(* Logix 5000 project; controller Hose_HP_Test_Rig_V1 vendor 1 type 14 code 149 rev 32.11; software revision 32.00; part 4 of 10 *)
(* tags used below, declared in another part *)
   BOTTOM_NOT_CLAMPED_STN3 : BOOL;
   DOOR_CLOSE_STS_STN2 : DINT;
   DOOR_CLOSE_STS_STN3 : DINT;
   DOOR_CLOSE_STS_STN4 : DINT;
   EXHS_OK_DEL_STN2 : TIMER;
   EXHS_OK_DELSTN4 : TIMER;
   EXHS_VAL_HP_ON_STN2 : BOOL;
   EXHS_VAL_OFF_CE_STN2 : BOOL;
   EXHS_VAL_OFF_CE_STN3 : BOOL;
   EXHS_VAL_OFF_TE_STN2 : BOOL;
   EXHS_VAL_OFF_TE_STN3 : BOOL;
   ONS28 : BOOL;
   ONS29 : BOOL;
   ONS30 : BOOL;
   ONS31 : BOOL;
   ONS32 : BOOL;
   ONS33 : BOOL;
   TOP_NOT_CLAMPED_STN2 : BOOL;
   TOP_NOT_CLAMPED_STN3 : BOOL;
   TOP_NOT_CLAMPED_STN4 : BOOL;
   ABORT_STN2 : BOOL;
   ABORT_STN3 : BOOL;
   ABORT_STN4 : BOOL;
   ACT_DROP_STN2 : REAL;
   ACT_DROP_STN3 : REAL;
   ACT_DROP_STN4 : REAL;
   ACT_PR_STN2 : REAL;
   ACT_PR_STN3 : REAL;
   ACT_PR_STN4 : REAL;
   AUTO_TEST_ON_STN2 : BOOL;
   AUTO_TEST_ON_STN3 : BOOL;
   AUTO_TEST_ON_STN4 : BOOL;
   BOTTOM_CLAMP_AUTO_STN2 : BOOL;
   BOTTOM_CLAMP_AUTO_STN3 : BOOL;
   BOTTOM_CLAMP_AUTO_STN4 : BOOL;
   BOTTOM_CLAMP_BLK_STN2 : DA_SOL_FWD_SEQ;
   BOTTOM_CLAMP_BLK_STN3 : DA_SOL_FWD_SEQ;
   BOTTOM_CLAMP_BLK_STN4 : DA_SOL_FWD_SEQ;
   BOTTOM_CLAMP_OK_STN1 : BOOL;
   BOTTOM_CLAMP_OK_STN3 : BOOL;
   BOTTOM_CLAMP_OK_STN4 : BOOL;
   BOTTOM_CLAMP_PS_STN2 : ALIAS FOR Local:2:I.Data.2;
   BOTTOM_CLAMP_PS_STN3 : ALIAS FOR Local:2:I.Data.7;
   BOTTOM_CLAMP_PS_STN4 : ALIAS FOR Local:2:I.Data.12;
   BOTTOM_CLAMP_SEQ_STN2 : DINT;
   BOTTOM_CLAMP_SEQ_STN3 : DINT;
   BOTTOM_CLAMP_SEQ_STN4 : DINT;
   BOTTOM_DECLAMP_AUTO_STN2 : BOOL;
   BOTTOM_DECLAMP_AUTO_STN3 : BOOL;
   BOTTOM_DECLAMP_AUTO_STN4 : BOOL;
   BOTTOM_DECLAMP_SEQ_STN2 : DINT;
   BOTTOM_DECLAMP_SEQ_STN3 : DINT;
   BOTTOM_DECLAMP_SEQ_STN4 : DINT;
   BOTTOM_DECLMP_BLK_STN2 : DA_SOL_RET_SEQ;
   BOTTOM_DECLMP_BLK_STN3 : DA_SOL_RET_SEQ;
   BOTTOM_DECLMP_BLK_STN4 : DA_SOL_RET_SEQ;
   BOTTOM_NOT_CLAMPED_STN2 : BOOL;
   BOTTOM_NOT_CLAMPED_STN4 : BOOL;
   BOTTOM_NOT_DECLAMPED_STN2 : BOOL;
   BOTTOM_NOT_DECLAMPED_STN3 : BOOL;
   BOTTOM_NOT_DECLAMPED_STN4 : BOOL;
   CHECK_TRACE_STS_STN2 : BOOL;
   CHECK_TRACE_STS_STN3 : BOOL;
   CHECK_TRACE_STS_STN4 : BOOL;
   CLR_FAIL_ONS_STN2 : BOOL;
   CLR_FAIL_ONS_STN3 : BOOL;
   CLR_FAIL_ONS_STN4 : BOOL;
   CLR_ONS_STN2 : BOOL;
   CLR_ONS_STN3 : BOOL;
   CLR_ONS_STN4 : BOOL;
   COMP_FAULT_STN2 : BOOL;
   COMP_FAULT_STN3 : BOOL;
   COMP_FAULT_STN4 : BOOL;
   CONS_CALB_ON_STN2 : BOOL;
   CONS_CALB_ON_STN3 : BOOL;
   CONS_CALB_ON_STN4 : BOOL;
   CONS_STS_STN2 : DINT;
   CONS_STS_STN4 : DINT;
   CONS_TEST_ON : BOOL;
   CONSTRICTION_TEST_ON_STN2 : BOOL;
   CONSTRICTION_TEST_ON_STN3 : BOOL;
   CONSTRICTION_TEST_ON_STN4 : BOOL;
   DICH_STN1 : INT;
   DOOR_CLOSE_ABORT_STN2 : BOOL;
   DOOR_CLOSE_ABORT_STN3 : BOOL;
   DOOR_CLOSE_ABORT_STN4 : BOOL;
   DOOR_CLOSE_AUTO_STN2 : BOOL;
   DOOR_CLOSE_AUTO_STN3 : BOOL;
   DOOR_CLOSE_AUTO_STN4 : BOOL;
   DOOR_CLOSE_BLK_STN2 : DOOR_CLOSE;
   DOOR_CLOSE_BLK_STN3 : DOOR_CLOSE;
   DOOR_CLOSE_BLK_STN4 : DOOR_CLOSE;
   DOOR_CLOSE_OK_STN2 : BOOL;
   DOOR_CLOSE_OK_STN3 : BOOL;
   DOOR_CLOSE_OK_STN4 : BOOL;
   DOOR_CLOSE_RS_STN2 : ALIAS FOR Local:2:I.Data.0;
   DOOR_CLOSE_RS_STN3 : ALIAS FOR Local:2:I.Data.5;
   DOOR_CLOSE_RS_STN4 : ALIAS FOR Local:2:I.Data.9;
   DOOR_CLOSE_SEQ_STN2 : DA_SOL_FWD_SEQ;
   DOOR_CLOSE_SEQ_STN3 : DA_SOL_FWD_SEQ;
   DOOR_CLOSE_SEQ_STN4 : DA_SOL_FWD_SEQ;
   DOOR_NOT_CLOSED_STN2 : BOOL;
   DOOR_NOT_CLOSED_STN3 : BOOL;
   DOOR_NOT_CLOSED_STN4 : BOOL;
   DOOR_OPEN_RS_STN2 : ALIAS FOR Local:1:I.Data.15;
   DOOR_OPEN_RS_STN3 : ALIAS FOR Local:2:I.Data.4;
   DOOR_OPEN_RS_STN4 : ALIAS FOR Local:2:I.Data.10;
   DROP_CHK_SEQ_STN2 : DROP_CHECK;
   DROP_CHK_SEQ_STN3 : DROP_CHECK;
   DROP_CHK_SEQ_STN4 : DROP_CHECK;
   DROP_NOK_STN2 : BOOL;
   DROP_NOK_STN3 : BOOL;
   DROP_NOK_STN4 : BOOL;
   DROP_OK_STN2 : BOOL;
   DROP_OK_STN3 : BOOL;
   DROP_OK_STN4 : BOOL;
   DUPLICATE_STN2 : BOOL;
   DUPLICATE_STN3 : BOOL;
   DUPLICATE_STN4 : BOOL;
   EC_STN1 : DINT;
   EC_STN2 : DINT;
   EC_STN3 : DINT;
   EC_STN4 : DINT;
   EXHAUST_SET_LIM : REAL;
   EXHS_OFF_BLK_STN2 : FILL_VAL_OFF;
   EXHS_OFF_BLK_STN3 : FILL_VAL_OFF;
   EXHS_OFF_BLK_STN4 : FILL_VAL_OFF;
   EXHS_OK_DEL_STN3 : TIMER;
   EXHS_VAL_HP_ON_STN3 : BOOL;
   EXHS_VAL_HP_ON_STN4 : BOOL;
   EXHS_VAL_OFF_CE_STN4 : BOOL;
   EXHS_VAL_OFF_STN2 : BOOL;
   EXHS_VAL_OFF_STN3 : BOOL;
   EXHS_VAL_OFF_STN4 : BOOL;
   EXHS_VAL_OFF_TE_STN4 : BOOL;
   FAULTED_STN2 : BOOL;
   FAULTED_STN3 : BOOL;
   FAULTED_STN4 : BOOL;
   FILL_ACT_TIME_STN2 : REAL;
   FILL_ACT_TIME_STN3 : REAL;
   FILL_ACT_TIME_STN4 : REAL;
   FILL_CHK_STN2 : PR_CHECK;
   FILL_CHK_STN3 : PR_CHECK;
   FILL_CHK_STN4 : PR_CHECK;
   FILL_HIGH_STN2 : BOOL;
   FILL_HIGH_STN3 : BOOL;
   FILL_HIGH_STN4 : BOOL;
   FILL_HL_STN1 : REAL;
   FILL_LL_STN1 : REAL;
   FILL_LOW_STN2 : BOOL;
   FILL_LOW_STN3 : BOOL;
   FILL_LOW_STN4 : BOOL;
   FILL_SEQ_START_STN2 : SEQ_START_AND_FILL;
   FILL_SEQ_START_STN3 : SEQ_START_AND_FILL;
   FILL_SEQ_START_STN4 : SEQ_START_AND_FILL;
   FILL_SET_TIME : REAL;
   FILL_VAL_OFF_SEQ_STN2 : FILL_VAL_OFF;
   FILL_VAL_OFF_SEQ_STN3 : FILL_VAL_OFF;
   FILL_VAL_OFF_SEQ_STN4 : FILL_VAL_OFF;
   FLT_CLR_ONS_STN2 : BOOL;
   FLT_CLR_ONS_STN3 : BOOL;
   FLT_CLR_ONS_STN4 : BOOL;
   HP_P2_STN2 : REAL;
   HP_P2_STN3 : REAL;
   HP_P2_STN4 : REAL;
   HP_STS_STN2 : DINT;
   HP_STS_STN3 : DINT;
   HP_STS_STN4 : DINT;
   HP_TEST_ON : BOOL;
   INCORRECT_STN2 : BOOL;
   INCORRECT_STN3 : BOOL;
   INCORRECT_STN4 : BOOL;
   INIT_STN2 : BOOL;
   INIT_STN3 : BOOL;
   INIT_STN4 : BOOL;
   LT_COMPLETED_STN2 : BOOL;
   LT_COMPLETED_STN3 : BOOL;
   LT_COMPLETED_STN4 : BOOL;
   LT_P1_STN2 : REAL;
   LT_P1_STN3 : REAL;
   LT_P1_STN4 : REAL;
   LT_POKEYOKE_STN2 : DINT;
   LT_POKEYOKE_STN3 : DINT;
   LT_POKEYOKE_STN4 : DINT;
   MSG_STN2 : DINT;
   MSG_STN3 : DINT;
   MSG_STN4 : DINT;
   P2_STN2 : REAL;
   P2_STN3 : REAL;
   P2_STN4 : REAL;
   POKEYOKE_NOT_DONE : BOOL;
   PYOKE_LT_STN2 : BOOL;
   PYOKE_LT_STN3 : BOOL;
   PYOKE_LT_STN4 : BOOL;
   RETEST : BOOL;
   RST_EXHS_VAL_OFF_STN2 : BOOL;
   RST_EXHS_VAL_OFF_STN3 : BOOL;
   RST_EXHS_VAL_OFF_STN4 : BOOL;
   RST_SEQ_ON_STN2 : BOOL;
   RST_SEQ_ON_STN3 : BOOL;
   RST_SEQ_ON_STN4 : BOOL;
   SCAN_OK_STN2 : BOOL;
   SCAN_OK_STN3 : BOOL;
   SCAN_OK_STN4 : BOOL;
   SCR_STS : DINT[6];
   SEQ_NO_STN2 : DINT;
   SEQ_NO_STN3 : DINT;
   SEQ_NO_STN4 : DINT;
   SET_DROP : REAL;
   STAB_ACT_TIME_STN2 : REAL;
   STAB_ACT_TIME_STN3 : REAL;
   STAB_ACT_TIME_STN4 : REAL;
   STAB_CHK_STN2 : PR_CHECK;
   STAB_CHK_STN3 : PR_CHECK;
   STAB_CHK_STN4 : PR_CHECK;
   STAB_HIGH_STN2 : BOOL;
   STAB_HIGH_STN3 : BOOL;
   STAB_HIGH_STN4 : BOOL;
   STAB_LOW_STN2 : BOOL;
   STAB_LOW_STN3 : BOOL;
   STAB_LOW_STN4 : BOOL;
   STAB_SET_TIME : REAL;
   STN2_ON : BOOL;
   STN3_ON : BOOL;
   STN4_ON : BOOL;
   TEST_ACT_TIME_STN2 : REAL;
   TEST_ACT_TIME_STN3 : REAL;
   TEST_ACT_TIME_STN4 : REAL;
   TEST_SET_TIME : REAL;
   TEST_STS_STN2 : DINT;
   TEST_STS_STN3 : DINT;
   TEST_STS_STN4 : DINT;
   TEST_STS_UPDATE_STN2 : TEST_TAIL_END;
   TEST_STS_UPDATE_STN3 : TEST_TAIL_END;
   TEST_STS_UPDATE_STN4 : TEST_TAIL_END;
   TEST_VAL_OFF_STN2 : BOOL;
   TEST_VAL_OFF_STN3 : BOOL;
   TEST_VAL_OFF_STN4 : BOOL;
   TEST_VAL_ON_STN2 : BOOL;
   TEST_VAL_ON_STN3 : BOOL;
   TEST_VAL_ON_STN4 : BOOL;
   TOP_CLAMP_AUTO_STN2 : BOOL;
   TOP_CLAMP_AUTO_STN3 : BOOL;
   TOP_CLAMP_AUTO_STN4 : BOOL;
   TOP_CLAMP_BLK_STN2 : DA_SOL_FWD_SEQ;
   TOP_CLAMP_BLK_STN3 : DA_SOL_FWD_SEQ;
   TOP_CLAMP_BLK_STN4 : DA_SOL_FWD_SEQ;
   TOP_CLAMP_OK_STN2 : BOOL;
   TOP_CLAMP_OK_STN3 : BOOL;
   TOP_CLAMP_OK_STN4 : BOOL;
(* MainProgram, continued *)

ROUTINE Auto_Test_Stn2   (* ladder *)
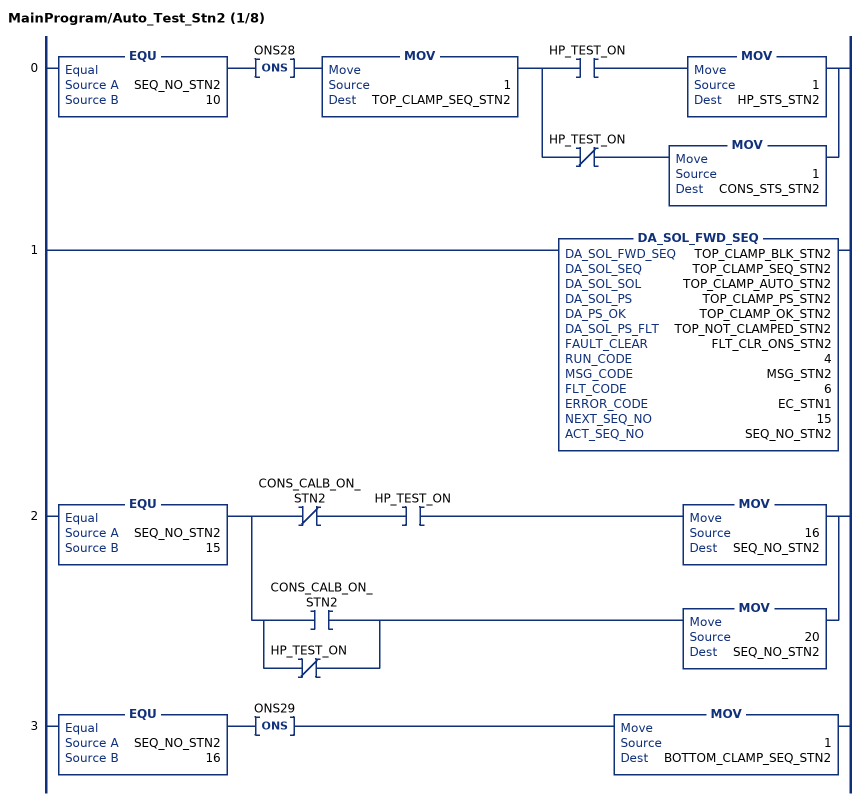
   0: EQU(SEQ_NO_STN2,10)ONS(ONS28)MOV(1,TOP_CLAMP_SEQ_STN2)[XIC(HP_TEST_ON) MOV(1,HP_STS_STN2) ,XIO(HP_TEST_ON) MOV(1,CONS_STS_STN2) ];
   1: DA_SOL_FWD_SEQ(TOP_CLAMP_BLK_STN2,TOP_CLAMP_SEQ_STN2,TOP_CLAMP_AUTO_STN2,TOP_CLAMP_PS_STN2,TOP_CLAMP_OK_STN2,TOP_NOT_CLAMPED_STN2,FLT_CLR_ONS_STN2,4,MSG_STN2,6,EC_STN1,15,SEQ_NO_STN2);
   2: EQU(SEQ_NO_STN2,15)[XIO(CONS_CALB_ON_STN2) XIC(HP_TEST_ON) MOV(16,SEQ_NO_STN2) ,[XIC(CONS_CALB_ON_STN2) ,XIO(HP_TEST_ON) ] MOV(20,SEQ_NO_STN2) ];
   3: EQU(SEQ_NO_STN2,16)ONS(ONS29)MOV(1,BOTTOM_CLAMP_SEQ_STN2);
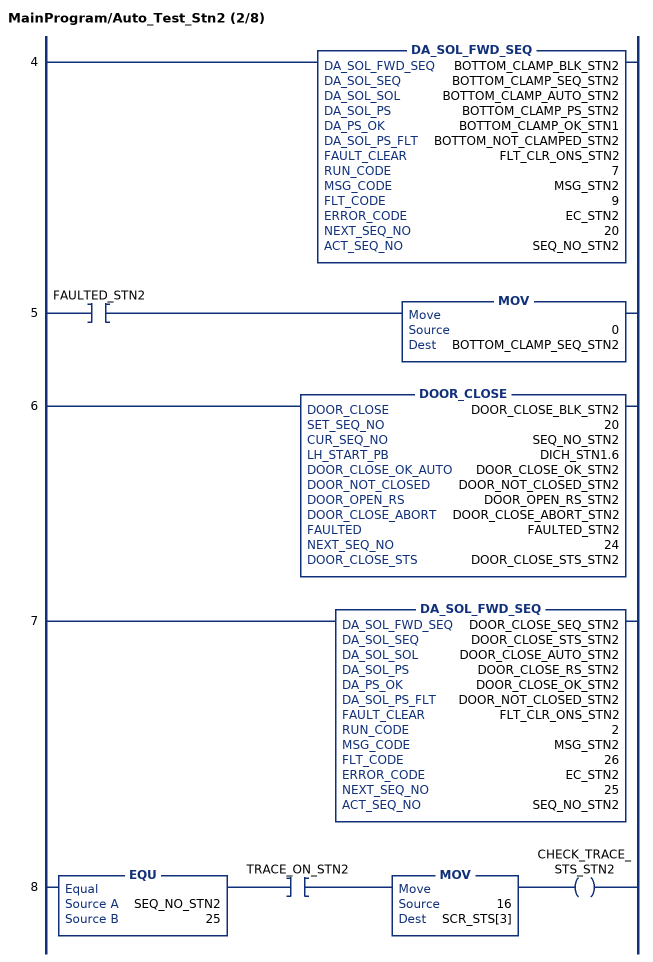
   4: DA_SOL_FWD_SEQ(BOTTOM_CLAMP_BLK_STN2,BOTTOM_CLAMP_SEQ_STN2,BOTTOM_CLAMP_AUTO_STN2,BOTTOM_CLAMP_PS_STN2,BOTTOM_CLAMP_OK_STN1,BOTTOM_NOT_CLAMPED_STN2,FLT_CLR_ONS_STN2,7,MSG_STN2,9,EC_STN2,20,SEQ_NO_STN2);
   5: XIC(FAULTED_STN2)MOV(0,BOTTOM_CLAMP_SEQ_STN2);
   6: DOOR_CLOSE(DOOR_CLOSE_BLK_STN2,20,SEQ_NO_STN2,DICH_STN1.6,DOOR_CLOSE_OK_STN2,DOOR_NOT_CLOSED_STN2,DOOR_OPEN_RS_STN2,DOOR_CLOSE_ABORT_STN2,FAULTED_STN2,24,DOOR_CLOSE_STS_STN2);
   7: DA_SOL_FWD_SEQ(DOOR_CLOSE_SEQ_STN2,DOOR_CLOSE_STS_STN2,DOOR_CLOSE_AUTO_STN2,DOOR_CLOSE_RS_STN2,DOOR_CLOSE_OK_STN2,DOOR_NOT_CLOSED_STN2,FLT_CLR_ONS_STN2,2,MSG_STN2,26,EC_STN2,25,SEQ_NO_STN2);
   8: EQU(SEQ_NO_STN2,25)XIC(TRACE_ON_STN2)MOV(16,SCR_STS[3])OTE(CHECK_TRACE_STS_STN2);
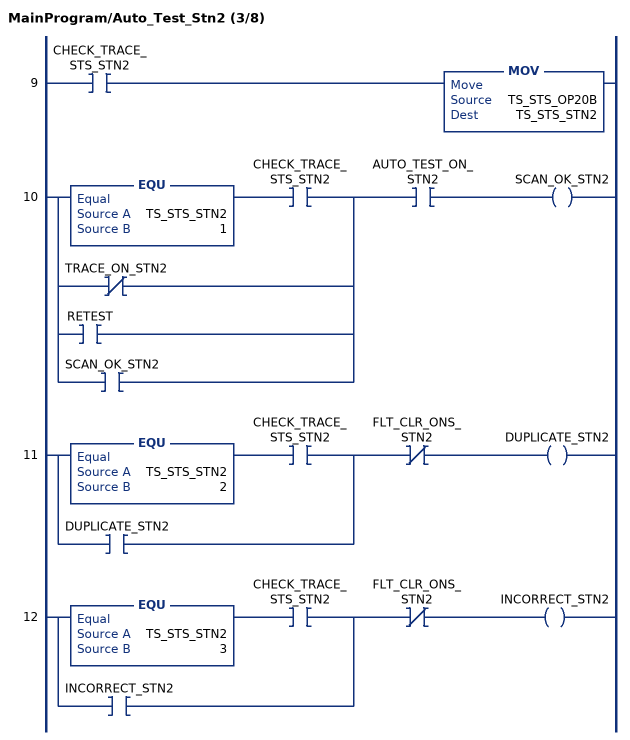
   9: XIC(CHECK_TRACE_STS_STN2)MOV(TS_STS_OP20B,TS_STS_STN2);
   10: [[EQU(TS_STS_STN2,1) XIC(CHECK_TRACE_STS_STN2) ,XIO(TRACE_ON_STN2) ,XIC(RETEST) ] ,XIC(SCAN_OK_STN2) ]XIC(AUTO_TEST_ON_STN2)OTE(SCAN_OK_STN2);
   11: [EQU(TS_STS_STN2,2) XIC(CHECK_TRACE_STS_STN2) ,XIC(DUPLICATE_STN2) ]XIO(FLT_CLR_ONS_STN2)OTE(DUPLICATE_STN2);
   12: [EQU(TS_STS_STN2,3) XIC(CHECK_TRACE_STS_STN2) ,XIC(INCORRECT_STN2) ]XIO(FLT_CLR_ONS_STN2)OTE(INCORRECT_STN2);
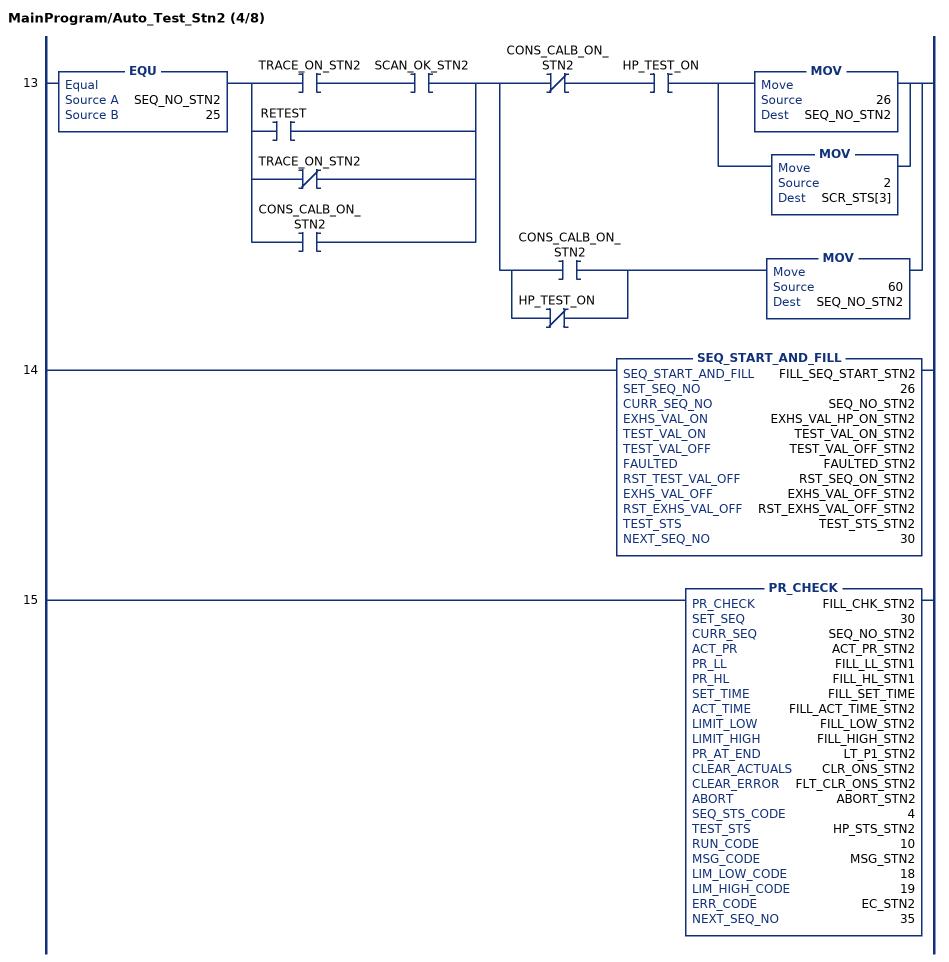
   13: EQU(SEQ_NO_STN2,25)[XIC(TRACE_ON_STN2) XIC(SCAN_OK_STN2) ,XIC(RETEST) ,XIO(TRACE_ON_STN2) ,XIC(CONS_CALB_ON_STN2) ][XIO(CONS_CALB_ON_STN2) XIC(HP_TEST_ON) [MOV(26,SEQ_NO_STN2) ,MOV(2,SCR_STS[3]) ] ,[XIC(CONS_CALB_ON_STN2) ,XIO(HP_TEST_ON) ] MOV(60,SEQ_NO_STN2) ];
   14: SEQ_START_AND_FILL(FILL_SEQ_START_STN2,26,SEQ_NO_STN2,EXHS_VAL_HP_ON_STN2,TEST_VAL_ON_STN2,TEST_VAL_OFF_STN2,FAULTED_STN2,RST_SEQ_ON_STN2,EXHS_VAL_OFF_STN2,RST_EXHS_VAL_OFF_STN2,TEST_STS_STN2,30);
   15: PR_CHECK(FILL_CHK_STN2,30,SEQ_NO_STN2,ACT_PR_STN2,FILL_LL_STN1,FILL_HL_STN1,FILL_SET_TIME,FILL_ACT_TIME_STN2,FILL_LOW_STN2,FILL_HIGH_STN2,LT_P1_STN2,CLR_ONS_STN2,FLT_CLR_ONS_STN2,ABORT_STN2,4,HP_STS_STN2,10,MSG_STN2,18,19,EC_STN2,35);
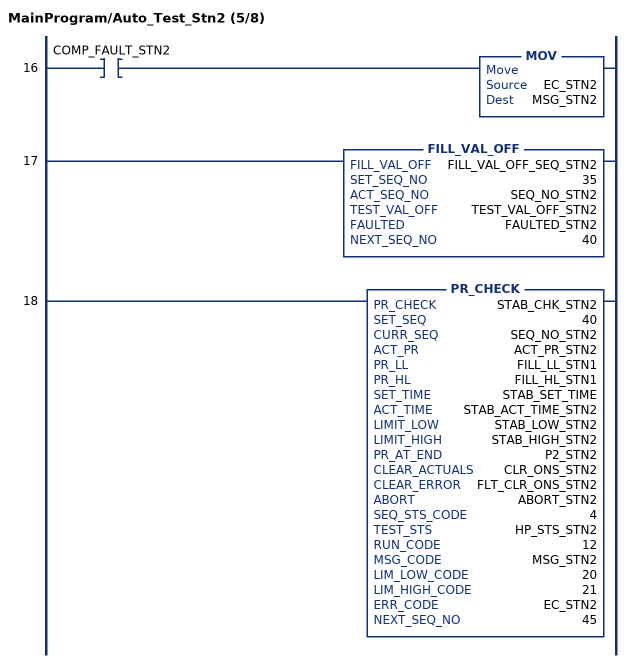
   16: XIC(COMP_FAULT_STN2)MOV(EC_STN2,MSG_STN2);
   17: FILL_VAL_OFF(FILL_VAL_OFF_SEQ_STN2,35,SEQ_NO_STN2,TEST_VAL_OFF_STN2,FAULTED_STN2,40);
   18: PR_CHECK(STAB_CHK_STN2,40,SEQ_NO_STN2,ACT_PR_STN2,FILL_LL_STN1,FILL_HL_STN1,STAB_SET_TIME,STAB_ACT_TIME_STN2,STAB_LOW_STN2,STAB_HIGH_STN2,P2_STN2,CLR_ONS_STN2,FLT_CLR_ONS_STN2,ABORT_STN2,4,HP_STS_STN2,12,MSG_STN2,20,21,EC_STN2,45);
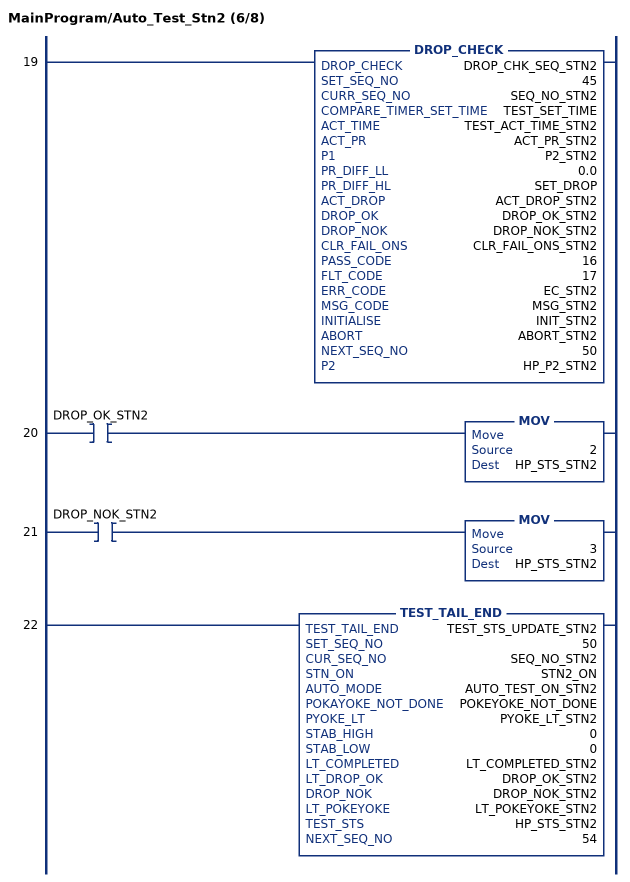
   19: DROP_CHECK(DROP_CHK_SEQ_STN2,45,SEQ_NO_STN2,TEST_SET_TIME,TEST_ACT_TIME_STN2,ACT_PR_STN2,P2_STN2,0.0,SET_DROP,ACT_DROP_STN2,DROP_OK_STN2,DROP_NOK_STN2,CLR_FAIL_ONS_STN2,16,17,EC_STN2,MSG_STN2,INIT_STN2,ABORT_STN2,50,HP_P2_STN2);
   20: XIC(DROP_OK_STN2)MOV(2,HP_STS_STN2);
   21: XIC(DROP_NOK_STN2)MOV(3,HP_STS_STN2);
   22: TEST_TAIL_END(TEST_STS_UPDATE_STN2,50,SEQ_NO_STN2,STN2_ON,AUTO_TEST_ON_STN2,POKEYOKE_NOT_DONE,PYOKE_LT_STN2,0,0,LT_COMPLETED_STN2,DROP_OK_STN2,DROP_NOK_STN2,LT_POKEYOKE_STN2,HP_STS_STN2,54);
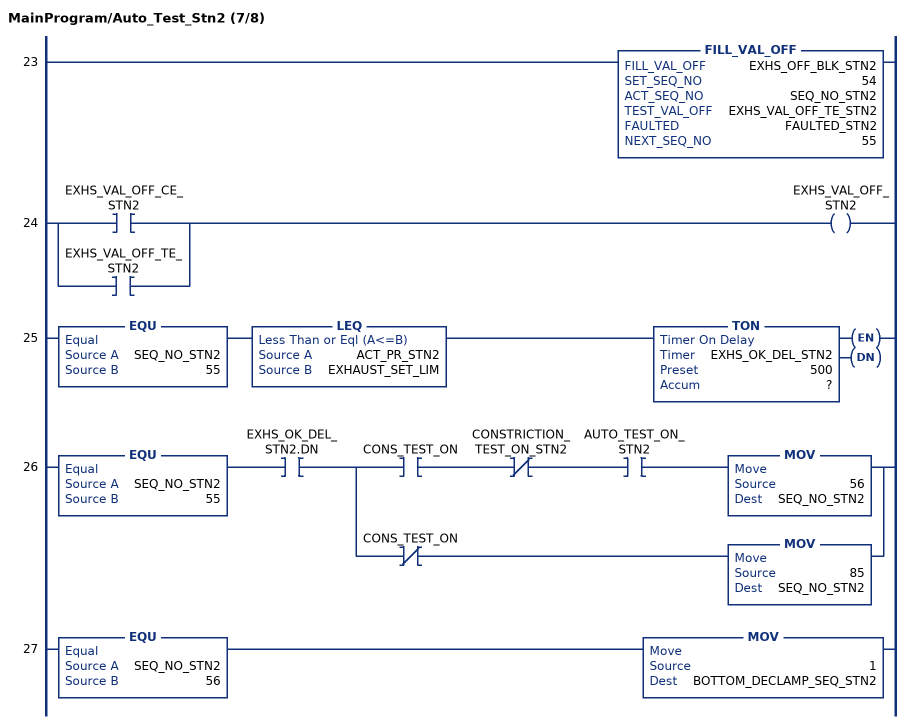
   23: FILL_VAL_OFF(EXHS_OFF_BLK_STN2,54,SEQ_NO_STN2,EXHS_VAL_OFF_TE_STN2,FAULTED_STN2,55);
   24: [XIC(EXHS_VAL_OFF_CE_STN2) ,XIC(EXHS_VAL_OFF_TE_STN2) ]OTE(EXHS_VAL_OFF_STN2);
   25: EQU(SEQ_NO_STN2,55)LEQ(ACT_PR_STN2,EXHAUST_SET_LIM)TON(EXHS_OK_DEL_STN2,?,?);
   26: EQU(SEQ_NO_STN2,55)XIC(EXHS_OK_DEL_STN2.DN)[XIC(CONS_TEST_ON) XIO(CONSTRICTION_TEST_ON_STN2) XIC(AUTO_TEST_ON_STN2) MOV(56,SEQ_NO_STN2) ,XIO(CONS_TEST_ON) MOV(85,SEQ_NO_STN2) ];
   27: EQU(SEQ_NO_STN2,56)MOV(1,BOTTOM_DECLAMP_SEQ_STN2);
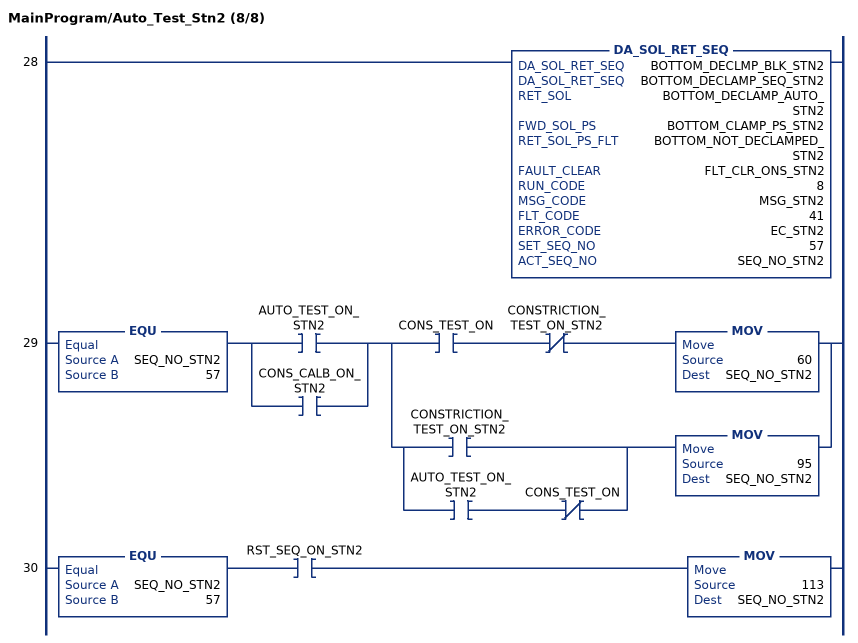
   28: DA_SOL_RET_SEQ(BOTTOM_DECLMP_BLK_STN2,BOTTOM_DECLAMP_SEQ_STN2,BOTTOM_DECLAMP_AUTO_STN2,BOTTOM_CLAMP_PS_STN2,BOTTOM_NOT_DECLAMPED_STN2,FLT_CLR_ONS_STN2,8,MSG_STN2,41,EC_STN2,57,SEQ_NO_STN2);
   29: EQU(SEQ_NO_STN2,57)[XIC(AUTO_TEST_ON_STN2) ,XIC(CONS_CALB_ON_STN2) ][XIC(CONS_TEST_ON) XIO(CONSTRICTION_TEST_ON_STN2) MOV(60,SEQ_NO_STN2) ,[XIC(CONSTRICTION_TEST_ON_STN2) ,XIC(AUTO_TEST_ON_STN2) XIO(CONS_TEST_ON) ] MOV(95,SEQ_NO_STN2) ];
   30: EQU(SEQ_NO_STN2,57)XIC(RST_SEQ_ON_STN2)MOV(113,SEQ_NO_STN2);
END_ROUTINE

ROUTINE Auto_Test_Stn3   (* ladder *)
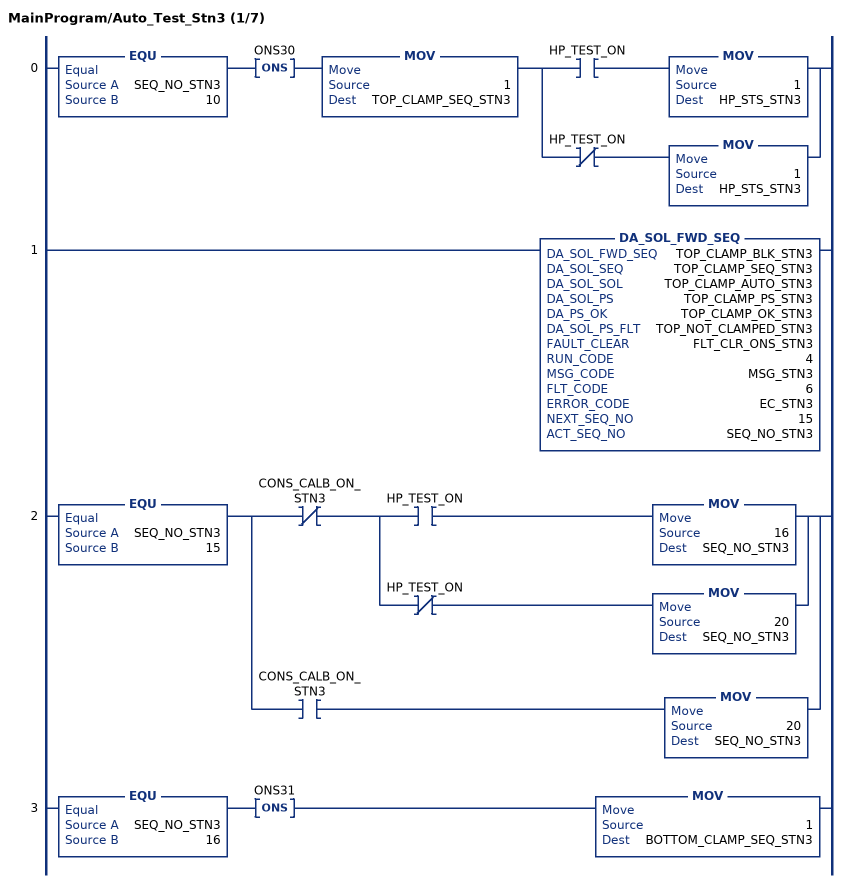
   0: EQU(SEQ_NO_STN3,10)ONS(ONS30)MOV(1,TOP_CLAMP_SEQ_STN3)[XIC(HP_TEST_ON) MOV(1,HP_STS_STN3) ,XIO(HP_TEST_ON) MOV(1,HP_STS_STN3) ];
   1: DA_SOL_FWD_SEQ(TOP_CLAMP_BLK_STN3,TOP_CLAMP_SEQ_STN3,TOP_CLAMP_AUTO_STN3,TOP_CLAMP_PS_STN3,TOP_CLAMP_OK_STN3,TOP_NOT_CLAMPED_STN3,FLT_CLR_ONS_STN3,4,MSG_STN3,6,EC_STN3,15,SEQ_NO_STN3);
   2: EQU(SEQ_NO_STN3,15)[XIO(CONS_CALB_ON_STN3) [XIC(HP_TEST_ON) MOV(16,SEQ_NO_STN3) ,XIO(HP_TEST_ON) MOV(20,SEQ_NO_STN3) ] ,XIC(CONS_CALB_ON_STN3) MOV(20,SEQ_NO_STN3) ];
   3: EQU(SEQ_NO_STN3,16)ONS(ONS31)MOV(1,BOTTOM_CLAMP_SEQ_STN3);
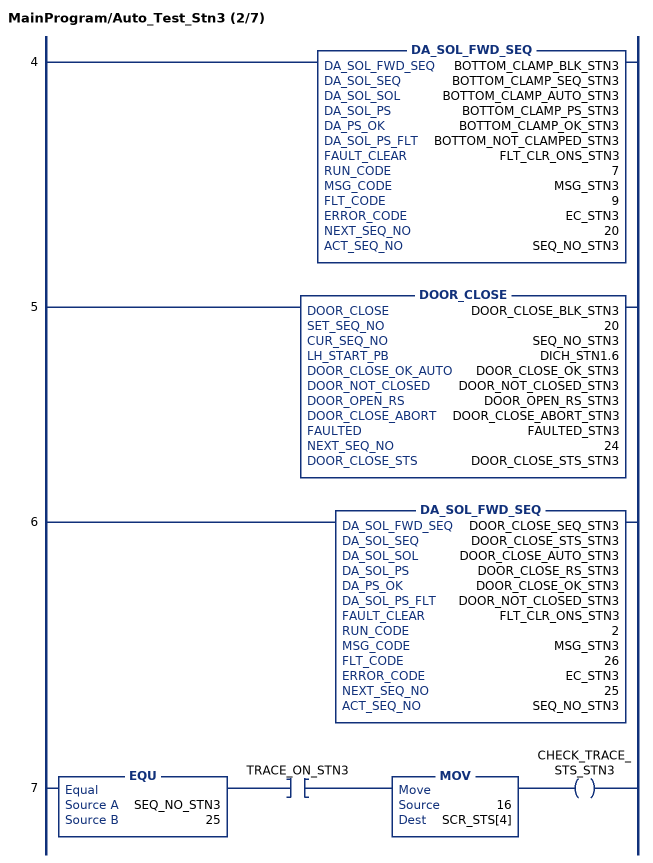
   4: DA_SOL_FWD_SEQ(BOTTOM_CLAMP_BLK_STN3,BOTTOM_CLAMP_SEQ_STN3,BOTTOM_CLAMP_AUTO_STN3,BOTTOM_CLAMP_PS_STN3,BOTTOM_CLAMP_OK_STN3,BOTTOM_NOT_CLAMPED_STN3,FLT_CLR_ONS_STN3,7,MSG_STN3,9,EC_STN3,20,SEQ_NO_STN3);
   5: DOOR_CLOSE(DOOR_CLOSE_BLK_STN3,20,SEQ_NO_STN3,DICH_STN1.6,DOOR_CLOSE_OK_STN3,DOOR_NOT_CLOSED_STN3,DOOR_OPEN_RS_STN3,DOOR_CLOSE_ABORT_STN3,FAULTED_STN3,24,DOOR_CLOSE_STS_STN3);
   6: DA_SOL_FWD_SEQ(DOOR_CLOSE_SEQ_STN3,DOOR_CLOSE_STS_STN3,DOOR_CLOSE_AUTO_STN3,DOOR_CLOSE_RS_STN3,DOOR_CLOSE_OK_STN3,DOOR_NOT_CLOSED_STN3,FLT_CLR_ONS_STN3,2,MSG_STN3,26,EC_STN3,25,SEQ_NO_STN3);
   7: EQU(SEQ_NO_STN3,25)XIC(TRACE_ON_STN3)MOV(16,SCR_STS[4])OTE(CHECK_TRACE_STS_STN3);
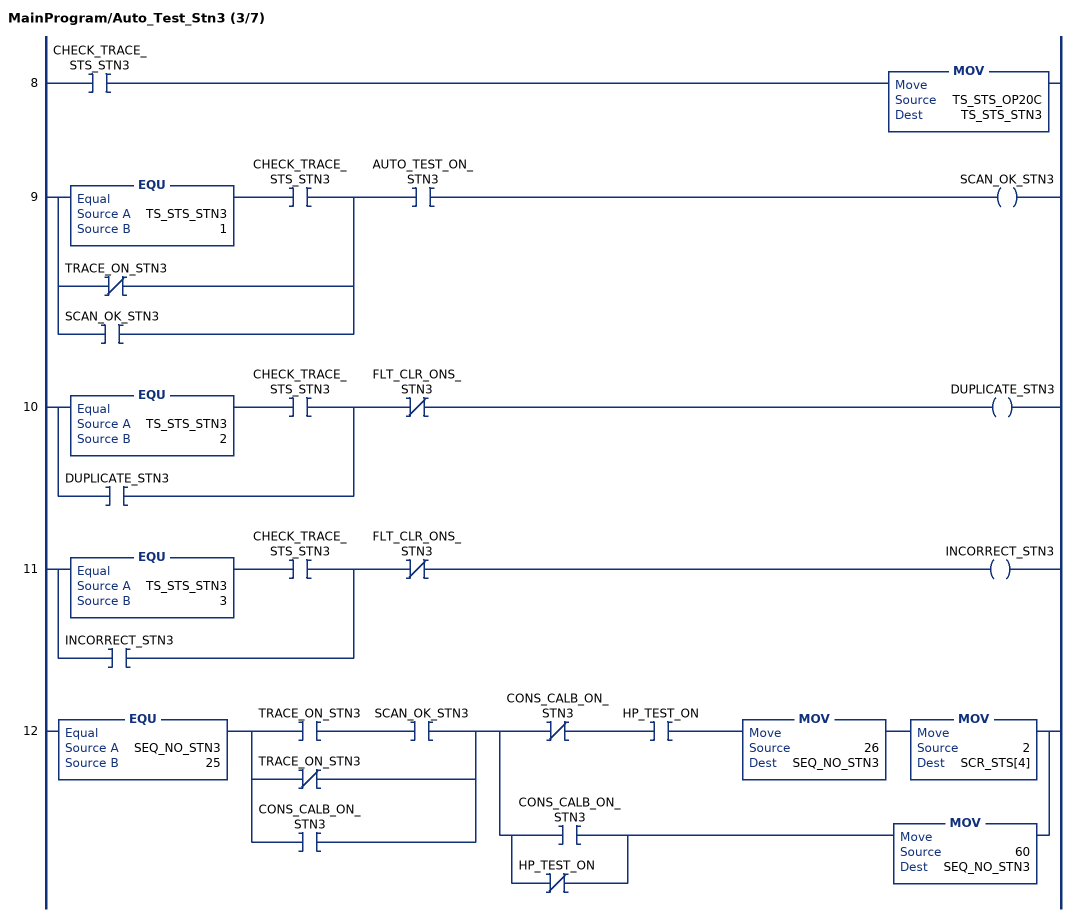
   8: XIC(CHECK_TRACE_STS_STN3)MOV(TS_STS_OP20C,TS_STS_STN3);
   9: [[EQU(TS_STS_STN3,1) XIC(CHECK_TRACE_STS_STN3) ,XIO(TRACE_ON_STN3) ] ,XIC(SCAN_OK_STN3) ]XIC(AUTO_TEST_ON_STN3)OTE(SCAN_OK_STN3);
   10: [EQU(TS_STS_STN3,2) XIC(CHECK_TRACE_STS_STN3) ,XIC(DUPLICATE_STN3) ]XIO(FLT_CLR_ONS_STN3)OTE(DUPLICATE_STN3);
   11: [EQU(TS_STS_STN3,3) XIC(CHECK_TRACE_STS_STN3) ,XIC(INCORRECT_STN3) ]XIO(FLT_CLR_ONS_STN3)OTE(INCORRECT_STN3);
   12: EQU(SEQ_NO_STN3,25)[XIC(TRACE_ON_STN3) XIC(SCAN_OK_STN3) ,XIO(TRACE_ON_STN3) ,XIC(CONS_CALB_ON_STN3) ][XIO(CONS_CALB_ON_STN3) XIC(HP_TEST_ON) MOV(26,SEQ_NO_STN3) MOV(2,SCR_STS[4]) ,[XIC(CONS_CALB_ON_STN3) ,XIO(HP_TEST_ON) ] MOV(60,SEQ_NO_STN3) ];
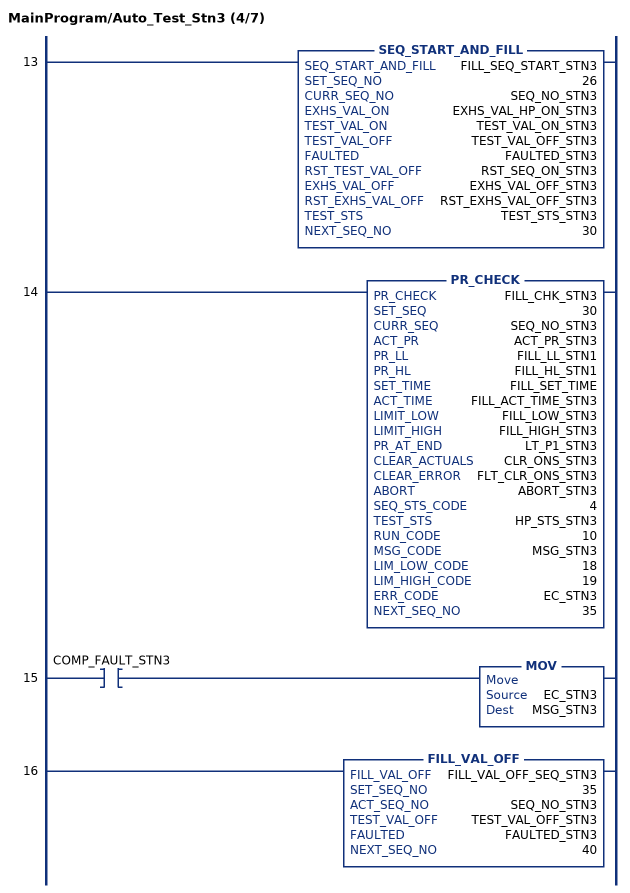
   13: SEQ_START_AND_FILL(FILL_SEQ_START_STN3,26,SEQ_NO_STN3,EXHS_VAL_HP_ON_STN3,TEST_VAL_ON_STN3,TEST_VAL_OFF_STN3,FAULTED_STN3,RST_SEQ_ON_STN3,EXHS_VAL_OFF_STN3,RST_EXHS_VAL_OFF_STN3,TEST_STS_STN3,30);
   14: PR_CHECK(FILL_CHK_STN3,30,SEQ_NO_STN3,ACT_PR_STN3,FILL_LL_STN1,FILL_HL_STN1,FILL_SET_TIME,FILL_ACT_TIME_STN3,FILL_LOW_STN3,FILL_HIGH_STN3,LT_P1_STN3,CLR_ONS_STN3,FLT_CLR_ONS_STN3,ABORT_STN3,4,HP_STS_STN3,10,MSG_STN3,18,19,EC_STN3,35);
   15: XIC(COMP_FAULT_STN3)MOV(EC_STN3,MSG_STN3);
   16: FILL_VAL_OFF(FILL_VAL_OFF_SEQ_STN3,35,SEQ_NO_STN3,TEST_VAL_OFF_STN3,FAULTED_STN3,40);
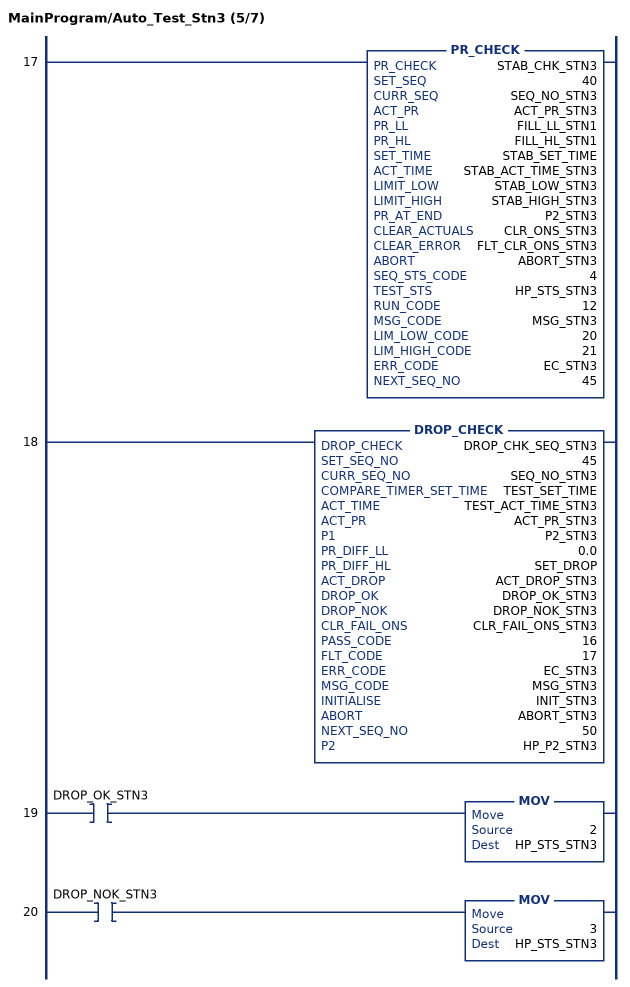
   17: PR_CHECK(STAB_CHK_STN3,40,SEQ_NO_STN3,ACT_PR_STN3,FILL_LL_STN1,FILL_HL_STN1,STAB_SET_TIME,STAB_ACT_TIME_STN3,STAB_LOW_STN3,STAB_HIGH_STN3,P2_STN3,CLR_ONS_STN3,FLT_CLR_ONS_STN3,ABORT_STN3,4,HP_STS_STN3,12,MSG_STN3,20,21,EC_STN3,45);
   18: DROP_CHECK(DROP_CHK_SEQ_STN3,45,SEQ_NO_STN3,TEST_SET_TIME,TEST_ACT_TIME_STN3,ACT_PR_STN3,P2_STN3,0.0,SET_DROP,ACT_DROP_STN3,DROP_OK_STN3,DROP_NOK_STN3,CLR_FAIL_ONS_STN3,16,17,EC_STN3,MSG_STN3,INIT_STN3,ABORT_STN3,50,HP_P2_STN3);
   19: XIC(DROP_OK_STN3)MOV(2,HP_STS_STN3);
   20: XIC(DROP_NOK_STN3)MOV(3,HP_STS_STN3);
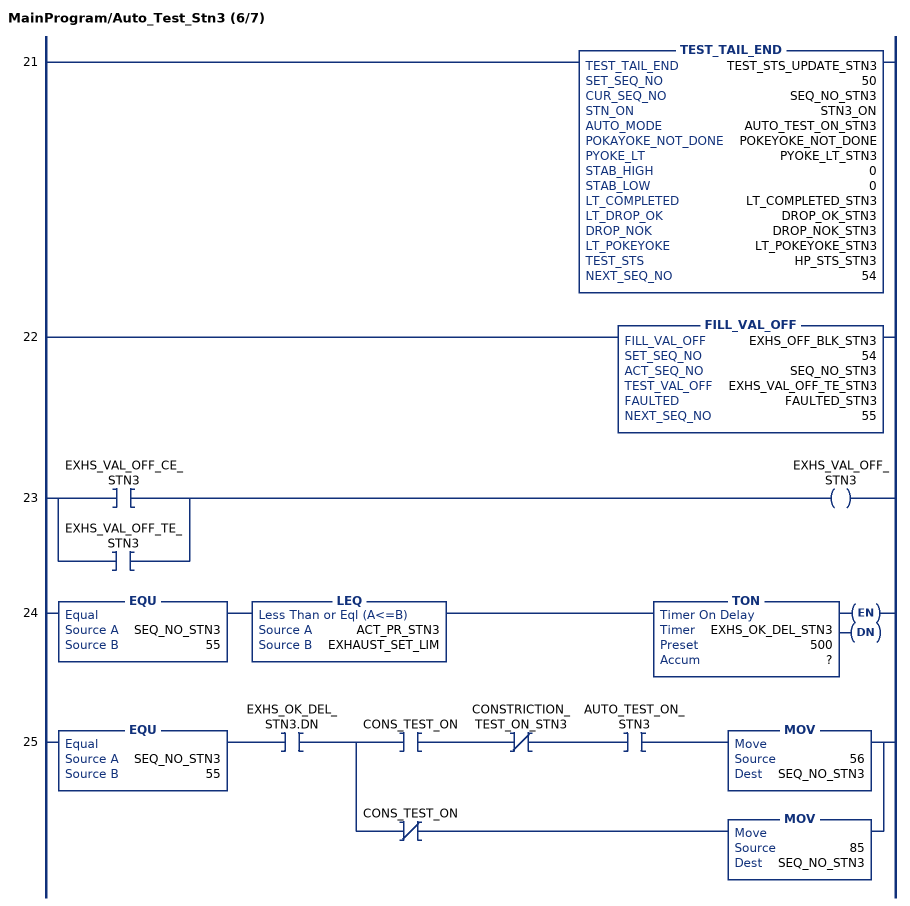
   21: TEST_TAIL_END(TEST_STS_UPDATE_STN3,50,SEQ_NO_STN3,STN3_ON,AUTO_TEST_ON_STN3,POKEYOKE_NOT_DONE,PYOKE_LT_STN3,0,0,LT_COMPLETED_STN3,DROP_OK_STN3,DROP_NOK_STN3,LT_POKEYOKE_STN3,HP_STS_STN3,54);
   22: FILL_VAL_OFF(EXHS_OFF_BLK_STN3,54,SEQ_NO_STN3,EXHS_VAL_OFF_TE_STN3,FAULTED_STN3,55);
   23: [XIC(EXHS_VAL_OFF_CE_STN3) ,XIC(EXHS_VAL_OFF_TE_STN3) ]OTE(EXHS_VAL_OFF_STN3);
   24: EQU(SEQ_NO_STN3,55)LEQ(ACT_PR_STN3,EXHAUST_SET_LIM)TON(EXHS_OK_DEL_STN3,?,?);
   25: EQU(SEQ_NO_STN3,55)XIC(EXHS_OK_DEL_STN3.DN)[XIC(CONS_TEST_ON) XIO(CONSTRICTION_TEST_ON_STN3) XIC(AUTO_TEST_ON_STN3) MOV(56,SEQ_NO_STN3) ,XIO(CONS_TEST_ON) MOV(85,SEQ_NO_STN3) ];
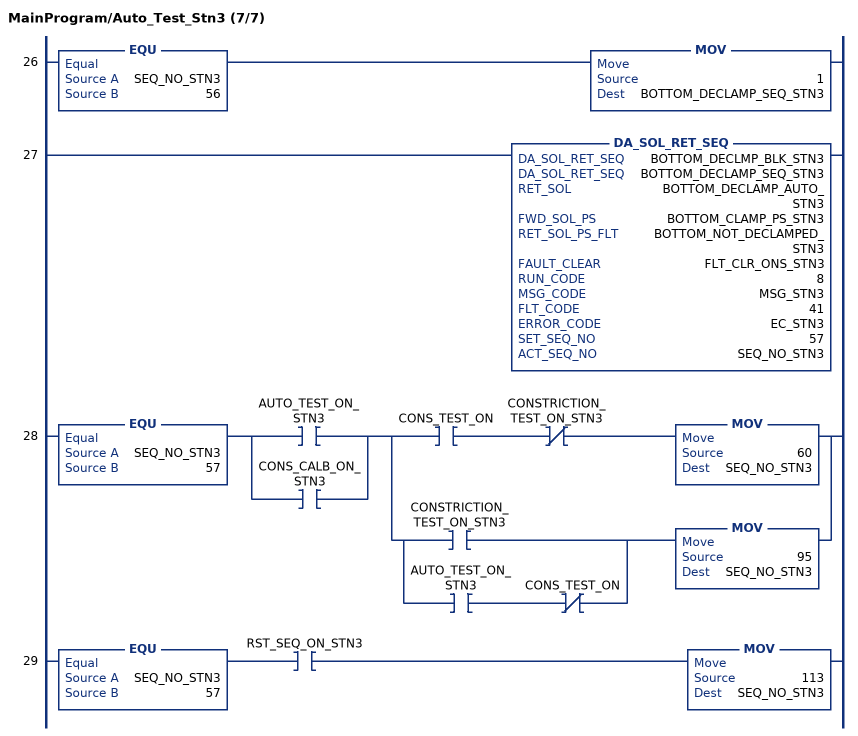
   26: EQU(SEQ_NO_STN3,56)MOV(1,BOTTOM_DECLAMP_SEQ_STN3);
   27: DA_SOL_RET_SEQ(BOTTOM_DECLMP_BLK_STN3,BOTTOM_DECLAMP_SEQ_STN3,BOTTOM_DECLAMP_AUTO_STN3,BOTTOM_CLAMP_PS_STN3,BOTTOM_NOT_DECLAMPED_STN3,FLT_CLR_ONS_STN3,8,MSG_STN3,41,EC_STN3,57,SEQ_NO_STN3);
   28: EQU(SEQ_NO_STN3,57)[XIC(AUTO_TEST_ON_STN3) ,XIC(CONS_CALB_ON_STN3) ][XIC(CONS_TEST_ON) XIO(CONSTRICTION_TEST_ON_STN3) MOV(60,SEQ_NO_STN3) ,[XIC(CONSTRICTION_TEST_ON_STN3) ,XIC(AUTO_TEST_ON_STN3) XIO(CONS_TEST_ON) ] MOV(95,SEQ_NO_STN3) ];
   29: EQU(SEQ_NO_STN3,57)XIC(RST_SEQ_ON_STN3)MOV(113,SEQ_NO_STN3);
END_ROUTINE

ROUTINE Auto_Test_Stn4   (* ladder *)
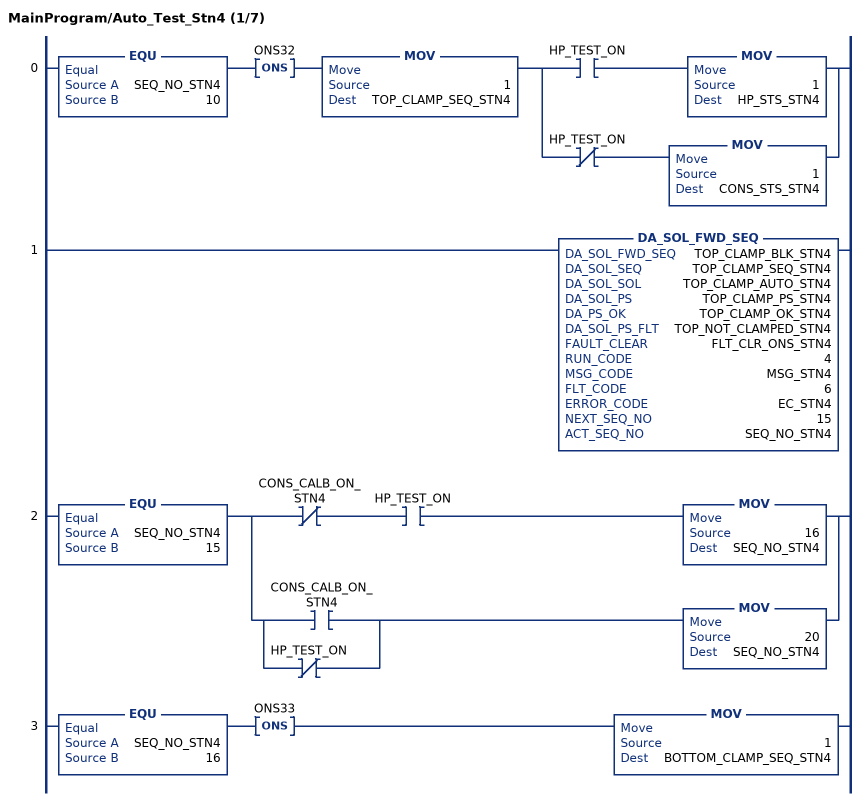
   0: EQU(SEQ_NO_STN4,10)ONS(ONS32)MOV(1,TOP_CLAMP_SEQ_STN4)[XIC(HP_TEST_ON) MOV(1,HP_STS_STN4) ,XIO(HP_TEST_ON) MOV(1,CONS_STS_STN4) ];
   1: DA_SOL_FWD_SEQ(TOP_CLAMP_BLK_STN4,TOP_CLAMP_SEQ_STN4,TOP_CLAMP_AUTO_STN4,TOP_CLAMP_PS_STN4,TOP_CLAMP_OK_STN4,TOP_NOT_CLAMPED_STN4,FLT_CLR_ONS_STN4,4,MSG_STN4,6,EC_STN4,15,SEQ_NO_STN4);
   2: EQU(SEQ_NO_STN4,15)[XIO(CONS_CALB_ON_STN4) XIC(HP_TEST_ON) MOV(16,SEQ_NO_STN4) ,[XIC(CONS_CALB_ON_STN4) ,XIO(HP_TEST_ON) ] MOV(20,SEQ_NO_STN4) ];
   3: EQU(SEQ_NO_STN4,16)ONS(ONS33)MOV(1,BOTTOM_CLAMP_SEQ_STN4);
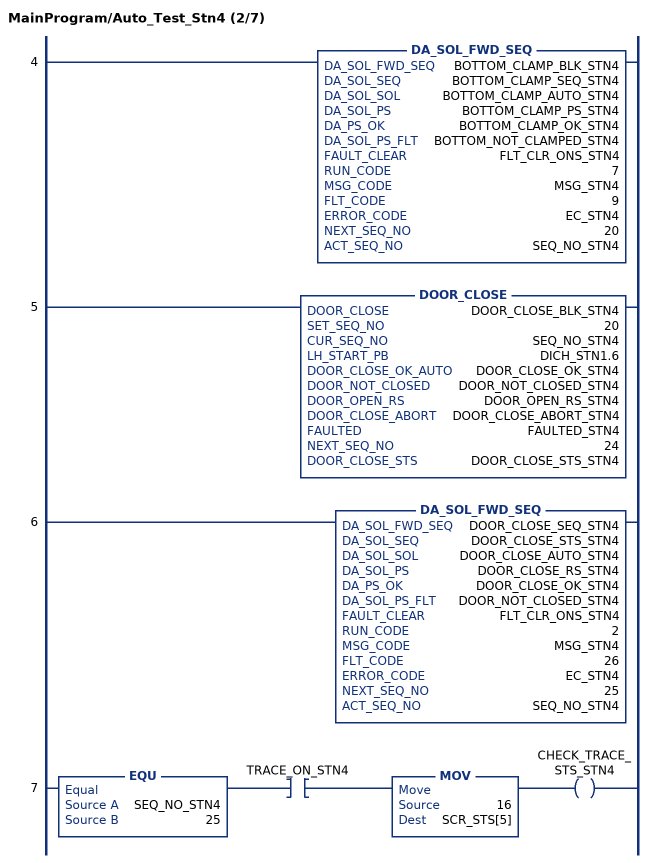
   4: DA_SOL_FWD_SEQ(BOTTOM_CLAMP_BLK_STN4,BOTTOM_CLAMP_SEQ_STN4,BOTTOM_CLAMP_AUTO_STN4,BOTTOM_CLAMP_PS_STN4,BOTTOM_CLAMP_OK_STN4,BOTTOM_NOT_CLAMPED_STN4,FLT_CLR_ONS_STN4,7,MSG_STN4,9,EC_STN4,20,SEQ_NO_STN4);
   5: DOOR_CLOSE(DOOR_CLOSE_BLK_STN4,20,SEQ_NO_STN4,DICH_STN1.6,DOOR_CLOSE_OK_STN4,DOOR_NOT_CLOSED_STN4,DOOR_OPEN_RS_STN4,DOOR_CLOSE_ABORT_STN4,FAULTED_STN4,24,DOOR_CLOSE_STS_STN4);
   6: DA_SOL_FWD_SEQ(DOOR_CLOSE_SEQ_STN4,DOOR_CLOSE_STS_STN4,DOOR_CLOSE_AUTO_STN4,DOOR_CLOSE_RS_STN4,DOOR_CLOSE_OK_STN4,DOOR_NOT_CLOSED_STN4,FLT_CLR_ONS_STN4,2,MSG_STN4,26,EC_STN4,25,SEQ_NO_STN4);
   7: EQU(SEQ_NO_STN4,25)XIC(TRACE_ON_STN4)MOV(16,SCR_STS[5])OTE(CHECK_TRACE_STS_STN4);
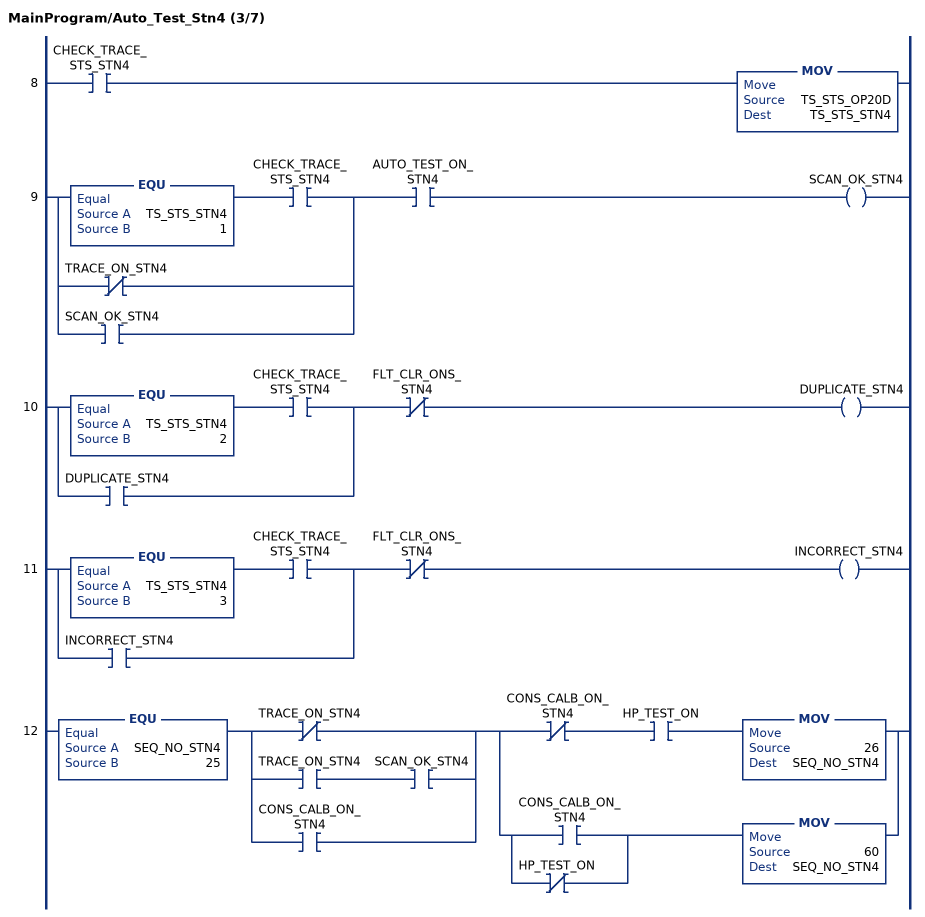
   8: XIC(CHECK_TRACE_STS_STN4)MOV(TS_STS_OP20D,TS_STS_STN4);
   9: [[EQU(TS_STS_STN4,1) XIC(CHECK_TRACE_STS_STN4) ,XIO(TRACE_ON_STN4) ] ,XIC(SCAN_OK_STN4) ]XIC(AUTO_TEST_ON_STN4)OTE(SCAN_OK_STN4);
   10: [EQU(TS_STS_STN4,2) XIC(CHECK_TRACE_STS_STN4) ,XIC(DUPLICATE_STN4) ]XIO(FLT_CLR_ONS_STN4)OTE(DUPLICATE_STN4);
   11: [EQU(TS_STS_STN4,3) XIC(CHECK_TRACE_STS_STN4) ,XIC(INCORRECT_STN4) ]XIO(FLT_CLR_ONS_STN4)OTE(INCORRECT_STN4);
   12: EQU(SEQ_NO_STN4,25)[XIO(TRACE_ON_STN4) ,XIC(TRACE_ON_STN4) XIC(SCAN_OK_STN4) ,XIC(CONS_CALB_ON_STN4) ][XIO(CONS_CALB_ON_STN4) XIC(HP_TEST_ON) MOV(26,SEQ_NO_STN4) ,[XIC(CONS_CALB_ON_STN4) ,XIO(HP_TEST_ON) ] MOV(60,SEQ_NO_STN4) ];
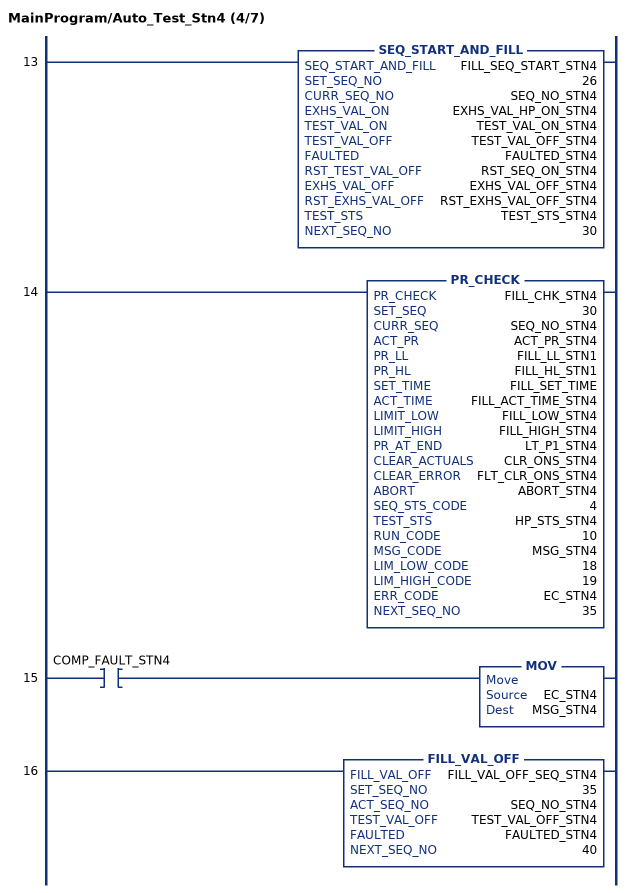
   13: SEQ_START_AND_FILL(FILL_SEQ_START_STN4,26,SEQ_NO_STN4,EXHS_VAL_HP_ON_STN4,TEST_VAL_ON_STN4,TEST_VAL_OFF_STN4,FAULTED_STN4,RST_SEQ_ON_STN4,EXHS_VAL_OFF_STN4,RST_EXHS_VAL_OFF_STN4,TEST_STS_STN4,30);
   14: PR_CHECK(FILL_CHK_STN4,30,SEQ_NO_STN4,ACT_PR_STN4,FILL_LL_STN1,FILL_HL_STN1,FILL_SET_TIME,FILL_ACT_TIME_STN4,FILL_LOW_STN4,FILL_HIGH_STN4,LT_P1_STN4,CLR_ONS_STN4,FLT_CLR_ONS_STN4,ABORT_STN4,4,HP_STS_STN4,10,MSG_STN4,18,19,EC_STN4,35);
   15: XIC(COMP_FAULT_STN4)MOV(EC_STN4,MSG_STN4);
   16: FILL_VAL_OFF(FILL_VAL_OFF_SEQ_STN4,35,SEQ_NO_STN4,TEST_VAL_OFF_STN4,FAULTED_STN4,40);
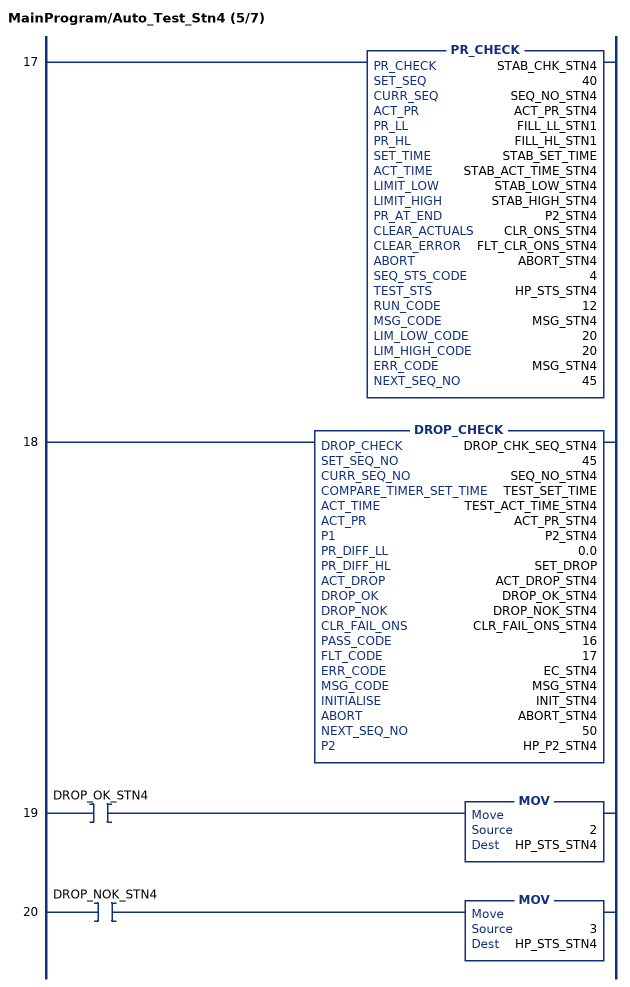
   17: PR_CHECK(STAB_CHK_STN4,40,SEQ_NO_STN4,ACT_PR_STN4,FILL_LL_STN1,FILL_HL_STN1,STAB_SET_TIME,STAB_ACT_TIME_STN4,STAB_LOW_STN4,STAB_HIGH_STN4,P2_STN4,CLR_ONS_STN4,FLT_CLR_ONS_STN4,ABORT_STN4,4,HP_STS_STN4,12,MSG_STN4,20,20,MSG_STN4,45);
   18: DROP_CHECK(DROP_CHK_SEQ_STN4,45,SEQ_NO_STN4,TEST_SET_TIME,TEST_ACT_TIME_STN4,ACT_PR_STN4,P2_STN4,0.0,SET_DROP,ACT_DROP_STN4,DROP_OK_STN4,DROP_NOK_STN4,CLR_FAIL_ONS_STN4,16,17,EC_STN4,MSG_STN4,INIT_STN4,ABORT_STN4,50,HP_P2_STN4);
   19: XIC(DROP_OK_STN4)MOV(2,HP_STS_STN4);
   20: XIC(DROP_NOK_STN4)MOV(3,HP_STS_STN4);
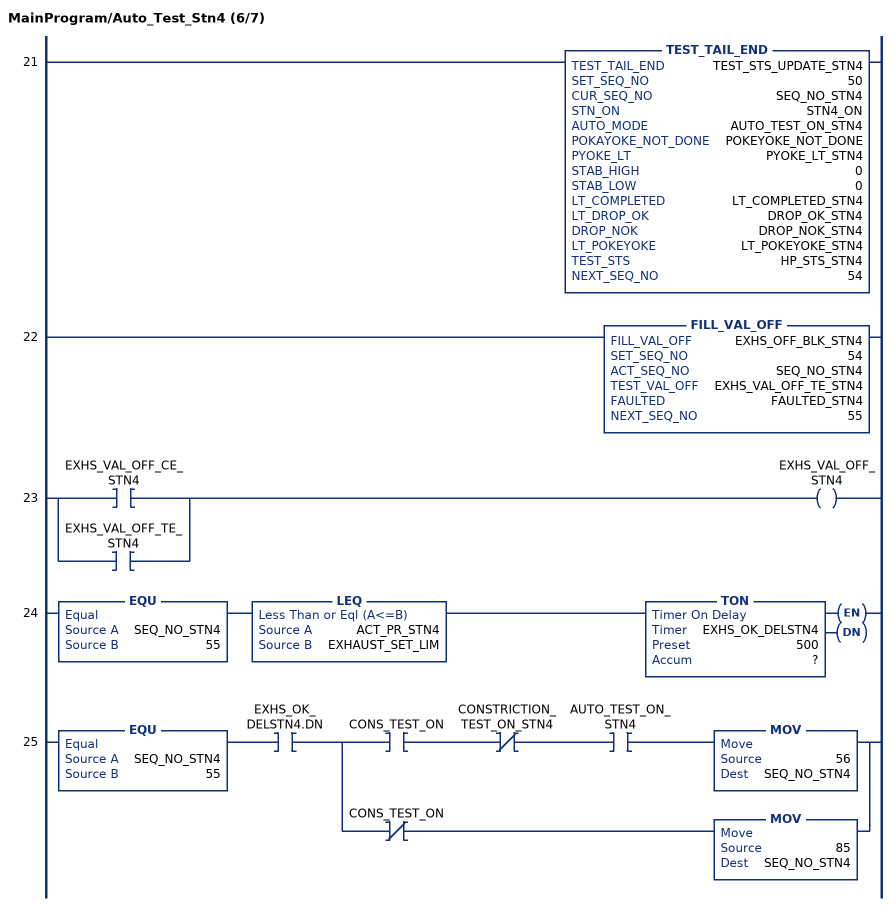
   21: TEST_TAIL_END(TEST_STS_UPDATE_STN4,50,SEQ_NO_STN4,STN4_ON,AUTO_TEST_ON_STN4,POKEYOKE_NOT_DONE,PYOKE_LT_STN4,0,0,LT_COMPLETED_STN4,DROP_OK_STN4,DROP_NOK_STN4,LT_POKEYOKE_STN4,HP_STS_STN4,54);
   22: FILL_VAL_OFF(EXHS_OFF_BLK_STN4,54,SEQ_NO_STN4,EXHS_VAL_OFF_TE_STN4,FAULTED_STN4,55);
   23: [XIC(EXHS_VAL_OFF_CE_STN4) ,XIC(EXHS_VAL_OFF_TE_STN4) ]OTE(EXHS_VAL_OFF_STN4);
   24: EQU(SEQ_NO_STN4,55)LEQ(ACT_PR_STN4,EXHAUST_SET_LIM)TON(EXHS_OK_DELSTN4,?,?);
   25: EQU(SEQ_NO_STN4,55)XIC(EXHS_OK_DELSTN4.DN)[XIC(CONS_TEST_ON) XIO(CONSTRICTION_TEST_ON_STN4) XIC(AUTO_TEST_ON_STN4) MOV(56,SEQ_NO_STN4) ,XIO(CONS_TEST_ON) MOV(85,SEQ_NO_STN4) ];
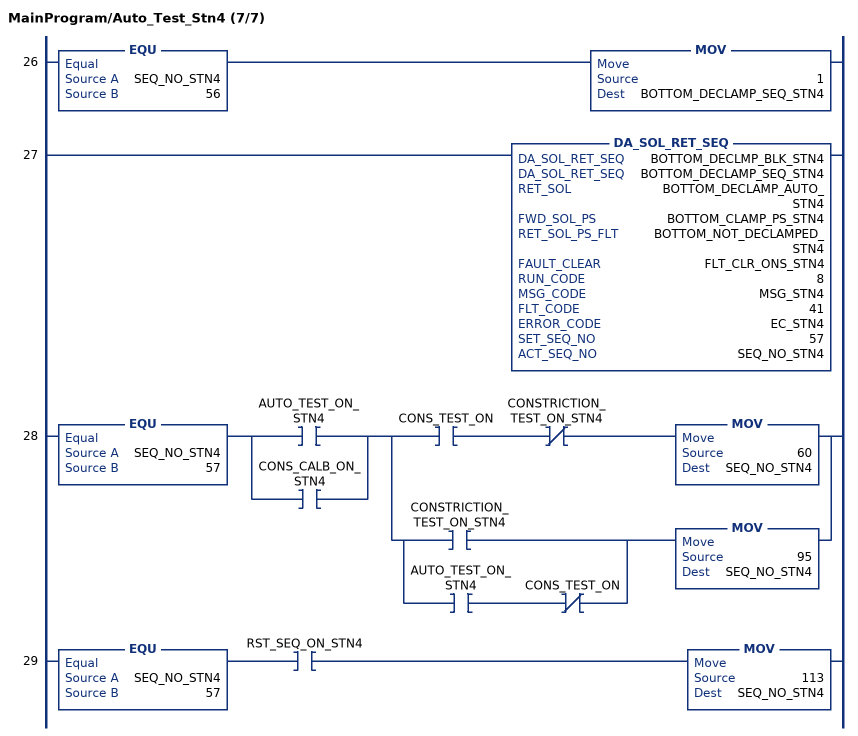
   26: EQU(SEQ_NO_STN4,56)MOV(1,BOTTOM_DECLAMP_SEQ_STN4);
   27: DA_SOL_RET_SEQ(BOTTOM_DECLMP_BLK_STN4,BOTTOM_DECLAMP_SEQ_STN4,BOTTOM_DECLAMP_AUTO_STN4,BOTTOM_CLAMP_PS_STN4,BOTTOM_NOT_DECLAMPED_STN4,FLT_CLR_ONS_STN4,8,MSG_STN4,41,EC_STN4,57,SEQ_NO_STN4);
   28: EQU(SEQ_NO_STN4,57)[XIC(AUTO_TEST_ON_STN4) ,XIC(CONS_CALB_ON_STN4) ][XIC(CONS_TEST_ON) XIO(CONSTRICTION_TEST_ON_STN4) MOV(60,SEQ_NO_STN4) ,[XIC(CONSTRICTION_TEST_ON_STN4) ,XIC(AUTO_TEST_ON_STN4) XIO(CONS_TEST_ON) ] MOV(95,SEQ_NO_STN4) ];
   29: EQU(SEQ_NO_STN4,57)XIC(RST_SEQ_ON_STN4)MOV(113,SEQ_NO_STN4);
END_ROUTINE
